Yaskawa INFORM job: R2_W27-A5(90,0)_MP_OK.JBI

/JOB
//NAME R2_W27-A5(90,0)_MP_OK
///FOLDERNAME MP_TEST
//POS
///NPOS 59,59,0,2,0,0
///TOOL 0
///POSTYPE PULSE
///PULSE
C00000=59274,-2798,-33333,-1733,105875,38300
C00001=56118,-55929,-65488,63507,82084,-79704
C00002=107302,11445,-18148,41871,56913,-66348
C00003=110741,32230,2763,42237,52953,-66643
C00004=120751,79647,39507,26761,71160,-57276
C00005=120751,79103,41400,26979,69865,-57588
C00006=120744,75848,38916,27042,69599,-57653
C00007=120744,78443,43396,27279,68325,-57966
C00008=118623,77776,52871,45412,57988,-54617
C00009=120750,88622,67725,49208,54909,-48496
C00010=120750,88631,67728,49206,54911,-48495
C00011=120750,88622,67725,49208,54909,-48496
C00012=120749,93703,83029,54455,33538,-41969
C00013=120749,91781,78018,51980,34828,-40628
C00014=120749,91783,78025,51984,34826,-40630
C00015=120749,91781,78018,51980,34828,-40628
C00016=116844,85517,70123,52684,38079,-41021
C00017=118789,65765,39976,46856,43765,-44990
C00018=111852,-24530,-46932,50155,56380,-74007
C00019=121112,34066,-5252,35562,63011,-58002
C00020=130011,57930,24474,30680,56437,-53277
C00021=134194,105572,72260,22632,68817,-46875
C00022=134194,105638,73419,22730,68188,-47002
C00023=134193,105753,74815,22850,67448,-47152
C00024=134194,105638,73419,22730,68188,-47002
C00025=134194,106258,78457,28233,60866,-48889
C00026=134193,106270,78464,28233,60867,-48888
C00027=134194,106258,78457,28233,60866,-48889
C00028=134190,113676,99568,26552,32426,-47426
C00029=134189,112987,98051,26153,32949,-47214
C00030=134189,112992,98062,26156,32945,-47216
C00031=134189,112987,98051,26153,32949,-47214
C00032=134190,113676,99568,26552,32426,-47426
C00033=134190,114038,100320,26747,32178,-47530
C00034=134190,113108,98381,26248,32821,-47265
C00035=132894,112231,98471,31075,32498,-48435
C00036=134187,61901,45630,36277,43695,-75561
C00037=134187,61910,45639,36278,43694,-75562
C00038=134187,61913,45643,36279,43693,-75562
C00039=133498,61457,45130,36693,44053,-75799
C00040=134183,61614,44049,35782,44371,-75250
C00041=134187,61913,45643,36279,43693,-75562
C00042=134187,61913,45643,36279,43693,-75562
C00043=134269,62376,46015,36219,43668,-75526
C00044=134187,61910,45639,36278,43694,-75562
C00045=134187,61901,45630,36277,43695,-75561
C00046=134187,61919,45650,29136,48325,-43573
C00047=134186,61925,45658,29136,48325,-43573
C00048=133508,61266,44910,29506,48668,-43803
C00049=133806,61307,43913,29055,49121,-43503
C00050=134186,61925,45657,29126,48327,-43573
C00051=134186,61925,45657,29126,48327,-43573
C00052=134187,61923,45655,29136,48325,-43573
C00053=129989,36005,23522,38083,39905,-49631
C00054=123209,5816,-13694,38205,48756,-49261
C00055=103853,-41691,-47930,50448,55954,-56439
C00056=56118,-55929,-65488,63507,82084,-79704
C00057=59274,-2798,-33333,-1733,105875,38300
C00058=59274,-2798,-33333,-1733,105875,38300
BC00000=158786,223116,705218
BC00001=216995,222898,12599
BC00002=216995,222898,12599
BC00003=216995,222898,12599
BC00004=218049,222894,53
BC00005=218049,222894,53
BC00006=210324,220573,53
BC00007=210324,220573,53
BC00008=221882,228945,53
BC00009=233503,237382,53
BC00010=231120,237215,53
BC00011=233503,237382,53
BC00012=212090,269672,53
BC00013=210567,269549,53
BC00014=210739,267251,53
BC00015=210567,269549,53
BC00016=210567,269549,53
BC00017=224162,251405,5940
BC00018=239220,185300,26771
BC00019=261727,224196,7509
BC00020=263734,233369,2370
BC00021=264639,237506,53
BC00022=262319,236808,53
BC00023=262303,236815,53
BC00024=262319,236808,53
BC00025=267458,243221,53
BC00026=265069,243229,53
BC00027=267458,243221,53
BC00028=256460,282614,53
BC00029=249382,282634,53
BC00030=249374,280330,53
BC00031=249382,282634,53
BC00032=256460,282614,53
BC00033=256431,275273,53
BC00034=258647,277099,53
BC00035=264190,281664,53
BC00036=266698,234070,100422
BC00037=261362,231476,82651
BC00038=259227,230438,75543
BC00039=259227,230438,75543
BC00040=259227,230438,75543
BC00041=259211,225830,75494
BC00042=259210,225397,75490
BC00043=259193,220789,75441
BC00044=261328,221826,82549
BC00045=266664,224420,100319
BC00046=260899,216913,95327
BC00047=258447,215444,90776
BC00048=258447,215444,90776
BC00049=258447,215444,90776
BC00050=258659,212473,90775
BC00051=258781,210847,90755
BC00052=259015,207877,90682
BC00053=259015,207877,90682
BC00054=259015,207877,90682
BC00055=259015,207877,90682
BC00056=216995,222898,12599
BC00057=158786,223116,705218
BC00058=158786,223116,705218
///POSTYPE BASE
///RECTAN
///RCONF 0,0,0,0,0,0,0,0,0,0,0,0,0,0,0,0,0,0,0,0,0,0,0,0
P00001=2714.263,6838.284,-998.276,27.8833,45.1566,-82.5967
P00006=0.222,-3.123,-1.508,0.0000,0.0000,0.0000
//INST
///DATE 2023/11/16 10:46
///ATTR SC,RW
///GROUP1 RB1,BS1
NOP
'r2_W27-A5(90,0)
'
'Path S848
SFTOF
MOVJ C00000 BC00000 VJ=20.00
MOVJ C00001 BC00001 VJ=20.00
MOVJ C00002 BC00002 VJ=20.00
MOVJ C00003 BC00003 VJ=20.00
MOVJ C00004 BC00004 VJ=20.00
MOVL C00005 BC00005 V=100.0
MOVL C00006 BC00006 V=100.0
REFP 3 C00007 BC00007
CALL JOB:SEARCH-R1
SET P001 P006
SFTON P001
MOVL C00008 BC00008 V=60.0
MOVL C00009 BC00009 V=60.0
REFP 3 C00010 BC00010
CALL JOB:SEARCH-R1
SET P001 P006
SFTON P001
MOVL C00011 BC00011 V=60.0
MOVL C00012 BC00012 V=100.0
MOVL C00013 BC00013 V=60.0
REFP 3 C00014 BC00014
CALL JOB:SEARCH-R1
SET P001 P006
SFTON P001
MOVL C00015 BC00015 V=60.0
MOVL C00016 BC00016 V=100.0
'Path VIA914
SFTOF
MOVJ C00017 BC00017 VJ=20.00
'Path VIA912
SFTOF
MOVJ C00018 BC00018 VJ=20.00
'Path VIA913
SFTOF
MOVJ C00019 BC00019 VJ=20.00
'Path S850
SFTOF
MOVJ C00020 BC00020 VJ=20.00
MOVL C00021 BC00021 V=100.0
MOVL C00022 BC00022 V=60.0
REFP 3 C00023 BC00023
CALL JOB:SEARCH-R1
SET P001 P006
SFTON P001
MOVL C00024 BC00024 V=60.0
MOVL C00025 BC00025 V=60.0
REFP 3 C00026 BC00026
CALL JOB:SEARCH-R1
SET P001 P006
SFTON P001
MOVL C00027 BC00027 V=60.0
MOVL C00028 BC00028 V=100.0
MOVL C00029 BC00029 V=60.0
REFP 3 C00030 BC00030
CALL JOB:SEARCH-R1
SET P001 P006
SFTON P001
MOVL C00031 BC00031 V=60.0
MOVL C00032 BC00032 V=100.0
MOVL C00033 BC00033 V=100.0
MOVL C00034 BC00034 V=100.0
MOVL C00035 BC00035 V=100.0
'Path W849
SFTOF
SFTON P001
MOVJ C00036 BC00036 VJ=20.00
MOVL C00037 BC00037 V=100.0
MOVL C00038 BC00038 V=100.0 PL=0
REFP 1 C00039 BC00039
REFP 2 C00040 BC00040
MACRO1 MJ#(0) ARGF7
COMM ARCON
MOVL C00041 BC00041 V=10.8
MOVL C00042 BC00042 V=10.8
MOVL C00043 BC00043 V=10.8
ARCOF
MOVL C00044 BC00044 V=100.0
MOVL C00045 BC00045 V=100.0
SFTOF
'Path W851
SFTOF
SFTON P001
MOVL C00046 BC00046 V=100.0
MOVL C00047 BC00047 V=100.0 PL=0
REFP 1 C00048 BC00048
REFP 2 C00049 BC00049
MACRO1 MJ#(0) ARGF7
ARCON
MOVL C00050 BC00050 V=10.8
MOVL C00051 BC00051 V=10.8
MOVL C00052 BC00052 V=10.8
ARCOF
MOVL C00053 BC00053 V=100.0
MOVJ C00054 BC00054 VJ=20.00
MOVJ C00055 BC00055 VJ=20.00
MOVJ C00056 BC00056 VJ=20.00
MOVJ C00057 BC00057 VJ=20.00
MOVJ C00058 BC00058 VJ=20.00
SFTOF
END
